// TIA Portal V19 export
DATA_BLOCK "_IOL_1Par_rd_wr_DATA"   // DB29
{ S7_Optimized_Access := 'TRUE' }
// stored: AutoNumber false, MemoryReserve 0
   VAR RETAIN
      ia : "_IOL_1Par_IA";   // ISDU Acyckic Single Parameter read / write data
      ihw_hwid : HW_ANY;   // Hardware Identifier of IO Master
      ii_cap : Int;   // Call Access Point
      ii_port : Int;   // Item connected to Port # of master
      i_datastorage : Bool;   // Activate Data Storage (IOL V1.1 devices only)
      i_blockparam : Bool;   // Activate Block Parameter Setting (IOL V1.1 devices only)
      iol_index : Int;   // Parameter decimal Index value
      iol_subindex : Int;   // Parameter decimal Sub-Index value
      len : Int;   // Read length in bytes
      o_comactiv : Bool;   // comms active
      io_fault : Bool;   // Fault
      io_rreq : Bool;   // Read request
      io_wreq : Bool;   // Write request
      io_reset : Bool;   // Fault Reset
   END_VAR
BEGIN
END_DATA_BLOCK
